% RSLogix 500 project I2P Hands-On 3 - Duncan.RSS, saved by version 10.00.00.00 %
PROJECT "ML01A"    % processor: Bul.1763 MicroLogix 1100 Series B %

PROGRAM FILES
  LAD 2   11 rungs

DATA FILES
  O0 OUTPUT  4 elements
  I1 INPUT  6 elements
  S2 STATUS  66 elements
  B3 BINARY  1 elements
  T4 TIMER  1 elements
  C5 COUNTER  1 elements
  R6 CONTROL  1 elements
  N7 INTEGER  1 elements
  F8 FLOAT  1 elements

LADDER 2
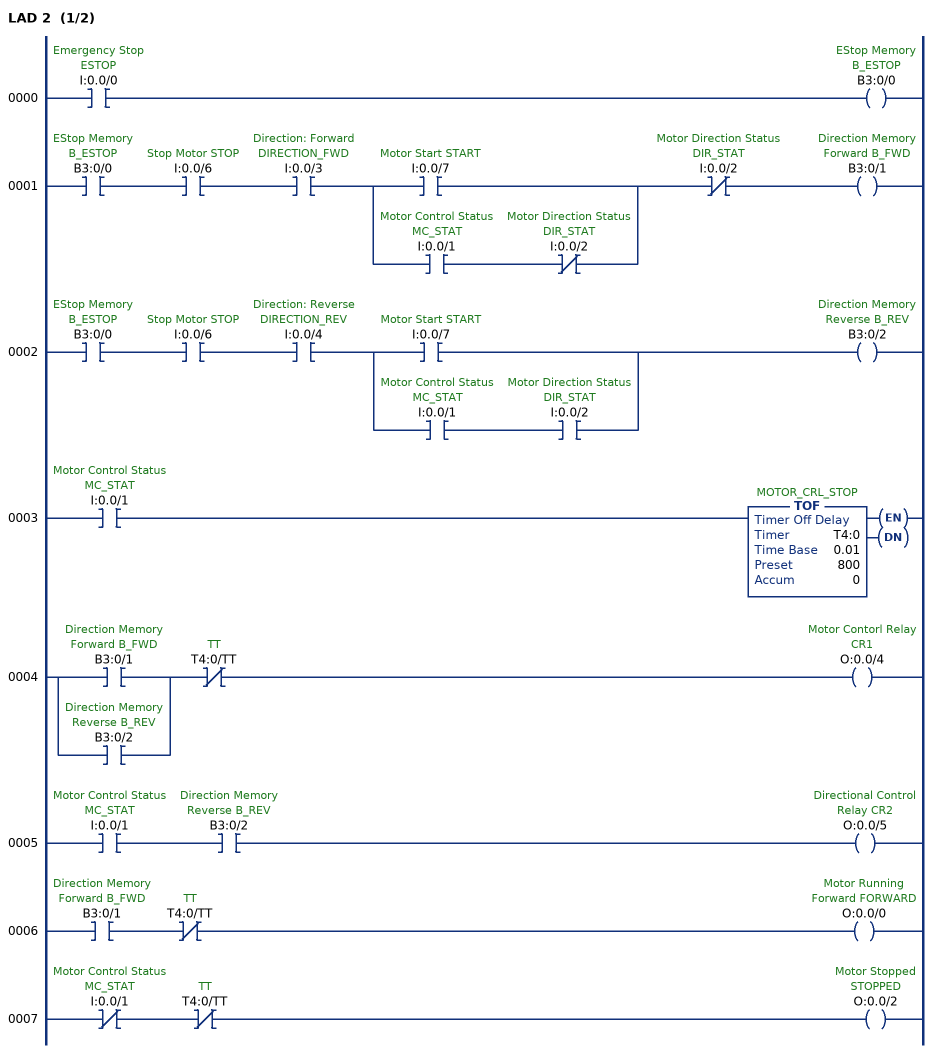
% Rung: 0 %
SOR XIC I:0.0/0 OTE B3:0/0 EOR
%   I:0.0/0  ESTOP  "Emergency Stop" %
%   B3:0/0  B_ESTOP  "EStop Memory" %
% Rung: 1 %
SOR XIC B3:0/0 XIC I:0.0/6 XIC I:0.0/3 BST XIC I:0.0/7 NXB XIC I:0.0/1 XIO I:0.0/2 BND XIO I:0.0/2 OTE B3:0/1 EOR
%   B3:0/0  B_ESTOP  "EStop Memory" %
%   I:0.0/6  STOP  "Stop Motor" %
%   I:0.0/3  DIRECTION_FWD  "Direction: Forward" %
%   I:0.0/7  START  "Motor Start" %
%   I:0.0/1  MC_STAT  "Motor Control Status" %
%   I:0.0/2  DIR_STAT  "Motor Direction Status" %
%   B3:0/1  B_FWD  "Direction Memory Forward" %
% Rung: 2 %
SOR XIC B3:0/0 XIC I:0.0/6 XIC I:0.0/4 BST XIC I:0.0/7 NXB XIC I:0.0/1 XIC I:0.0/2 BND OTE B3:0/2 EOR
%   B3:0/0  B_ESTOP  "EStop Memory" %
%   I:0.0/6  STOP  "Stop Motor" %
%   I:0.0/4  DIRECTION_REV  "Direction: Reverse" %
%   I:0.0/7  START  "Motor Start" %
%   I:0.0/1  MC_STAT  "Motor Control Status" %
%   I:0.0/2  DIR_STAT  "Motor Direction Status" %
%   B3:0/2  B_REV  "Direction Memory Reverse" %
% Rung: 3 %
SOR XIC I:0.0/1 TOF T4:0 0.01 800 0 EOR
%   I:0.0/1  MC_STAT  "Motor Control Status" %
%   T4:0  MOTOR_CRL_STOP %
% Rung: 4 %
SOR BST XIC B3:0/1 NXB XIC B3:0/2 BND XIO T4:0/TT OTE O:0.0/4 EOR
%   B3:0/1  B_FWD  "Direction Memory Forward" %
%   B3:0/2  B_REV  "Direction Memory Reverse" %
%   T4:0/TT  TT %
%   O:0.0/4  CR1  "Motor Contorl Relay" %
% Rung: 5 %
SOR XIC I:0.0/1 XIC B3:0/2 OTE O:0.0/5 EOR
%   I:0.0/1  MC_STAT  "Motor Control Status" %
%   B3:0/2  B_REV  "Direction Memory Reverse" %
%   O:0.0/5  CR2  "Directional Control Relay" %
% Rung: 6 %
SOR XIC B3:0/1 XIO T4:0/TT OTE O:0.0/0 EOR
%   B3:0/1  B_FWD  "Direction Memory Forward" %
%   T4:0/TT  TT %
%   O:0.0/0  FORWARD  "Motor Running Forward" %
% Rung: 7 %
SOR XIO I:0.0/1 XIO T4:0/TT OTE O:0.0/2 EOR
%   I:0.0/1  MC_STAT  "Motor Control Status" %
%   T4:0/TT  TT %
%   O:0.0/2  STOPPED  "Motor Stopped" %

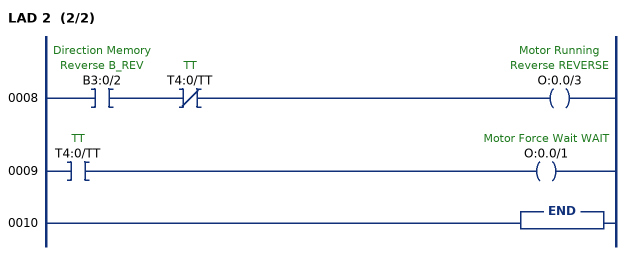
% Rung: 8 %
SOR XIC B3:0/2 XIO T4:0/TT OTE O:0.0/3 EOR
%   B3:0/2  B_REV  "Direction Memory Reverse" %
%   T4:0/TT  TT %
%   O:0.0/3  REVERSE  "Motor Running Reverse" %
% Rung: 9 %
SOR XIC T4:0/TT OTE O:0.0/1 EOR
%   T4:0/TT  TT %
%   O:0.0/1  WAIT  "Motor Force Wait" %
% Rung: 10 %
SOR END EOR

DATA TABLE (non-zero values as saved)
DATA B3
% B3:0 % 0X0001
DATA T4
% .PRE .ACC %
% T4:0 % 800 0
